
// ===== library: MasterCopy "maniobra_pintado" =====

FUNCTION_BLOCK "maniobra_pintado"   // FB6, STL
{ S7_Optimized_Access := 'TRUE' }
VERSION : 0.1
BEGIN
END_FUNCTION_BLOCK

// ===== library: MasterCopy "maniobra_grabado" =====

FUNCTION_BLOCK "maniobra_grabado"   // FB5, STL
{ S7_Optimized_Access := 'TRUE' }
VERSION : 0.1
BEGIN
END_FUNCTION_BLOCK